//{attribute 'qualified_only'}
{attribute 'strict'}
TYPE E_MessageIds :
(
	NoMessage_00 := 0,
	TransportCommand_05 := 5,
	LocationUpdateResponse_07 := 7,
	EquipmentStatusResponse_08 := 8,
	KeepAlive_09 := 9,
	Arrival_23 := 23,
	TransportResponse_25 := 25,
	TransportComplete_26 := 26,
	LocationUpdate_27 := 27,
	EquipmentStatusUpdate_28 := 28,
	KeepAliveResponse_29 := 29
);
END_TYPE

(* stored: Version 1.1.0.1, ProductVersion 3.1.4024.4
   EnumerationTextList E_MessageIds: Id {0e253860-a70b-46ad-9708-05ab49108d8c} *)
